# EPICS substitutions: iocBoot/ioc-xpp-gige-cam2/ioc-xpp-gige-cam2.substitutions
# IOC archive file
## Replace XPP:IOC:GIGE:02 with the PV prefix used for
## iocAdmin PV's on this IOC

# Generate IOC archive request
file archive_gige.archive
{
	{ IOC = "XPP:IOC:GIGE:02" }
}
